PROGRAM AutoExtrusion
VAR
END_VAR

END_PROGRAM

(* stored: Version 1.1.0.1, ProductVersion 3.1.4024.9
   POU AutoExtrusion: Id {86502c01-c062-40ed-a59d-dbd5307352d9}, SpecialFunc None *)
